FUNCTION_BLOCK E_SELECT (* selection between two events based on boolean input G *)
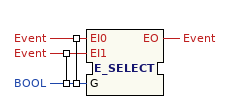
  EVENT_INPUT
    EI0 WITH G; (* Input event, selected when G=0 *)
    EI1 WITH G; (* Input event, selected when G=1 *)
  END_EVENT
  EVENT_OUTPUT
    EO; (* Output Event *)
  END_EVENT
  VAR_INPUT
    G : BOOL; (* Select EI0 when G=0, EI1 when G=1 *)
  END_VAR
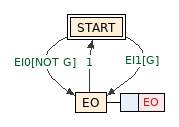
  EC_STATES
    START; (* Initial State *)
    EO : -> EO; (* Issue Output Event *)
  END_STATES
  EC_TRANSITIONS
    EO TO START := 1;
    START TO EO := EI0[NOT G];
    START TO EO := EI1[G];
  END_TRANSITIONS
END_FUNCTION_BLOCK
